Fanuc KAREL source: kb00188.KL

PROGRAM KB00188
%NOLOCKGROUP
VAR
P1 : STRING[80];RESULT:INTEGER
BEGIN
--
P1='A'
RESULT=STR_LEN(P1)
END KB00188
